// ---- POUs/P70_Interface.TcPOU
PROGRAM P70_Interface
VAR
END_VAR

(* UI Right Dashboard Variable*)
GVL_IO.aInputState[1].0 	:= GVL_IO.aDigitalInputIO[1].0; //Maintenance Key

// GVL_IO.aInputState[1].1		:= P92_Maintenance.bReactorCabinetLamp; //Reactor Cabinet Lamp
// GVL_IO.aInputState[1].2		:= P92_Maintenance.bGasCabinetLamp; // Gas Cabinet Lamp
// GVL_IO.aInputState[1].3		:= P92_Maintenance.bPowerDistributeLamp; // Power Cabinet Lamp
GVL_IO.aInputState[1].1		:= GVL_IO.aDigitalOutputIO[2].5; //Reactor Cabinet Lamp
GVL_IO.aInputState[1].2		:= GVL_IO.aDigitalOutputIO[2].6; // Gas Cabinet Lamp
GVL_IO.aInputState[1].3		:= GVL_IO.aDigitalOutputIO[2].7; // Power Cabinet Lamp

GVL_IO.aInputState[1].4 	:= GVL_IO.aDigitalInputIO[2].0; //CDA Alarm Switch
GVL_IO.aInputState[1].5		:= GVL_IO.aDigitalInputIO[2].1; //Water Flow Sensor

// GVL_IO.aInputState[1].6 	:= P11_E3508.isHeaterReady; //Induction Heater
// GVL_IO.aInputState[1].7 	:= P11_E3508.isHeaterRun; //Induction Heater
// GVL_IO.aInputState[1].8 	:= P11_E3508.isHeaterFault; //Induction Heater
GVL_IO.aInputState[1].6 	:= GVL_IO.aDigitalInputIO[2].2; //Induction Heater
GVL_IO.aInputState[1].7 	:= GVL_IO.aDigitalInputIO[2].3; //Induction Heater
GVL_IO.aInputState[1].8 	:= GVL_IO.aDigitalInputIO[2].4; //Induction Heater

// GVL_IO.aInputState[1].9	:= P15_RotationOperation.bStart_Stop; //Susceptor Rotation Motor
// GVL_IO.aInputState[1].10	:= P15_RotationOperation.bBrake_Run; //Susceptor Rotation Motor
// GVL_IO.aInputState[1].11	:= P15_RotationOperation.isRotationFault; //Susceptor Rotation Motor
GVL_IO.aInputState[1].9		:= GVL_IO.aDigitalOutputIO[3].4; //Susceptor Rotation Motor
GVL_IO.aInputState[1].10	:= GVL_IO.aDigitalOutputIO[3].5; //Susceptor Rotation Motor

// GVL_IO.aInputState[1].12 	:= P12_IQ_PLUS.isPumpWarning; //Vacuum Pump
// GVL_IO.aInputState[1].13 	:= P12_IQ_PLUS.isPumpRunning; //Vacuum Pump
// GVL_IO.aInputState[1].14 	:= P12_IQ_PLUS.isPumpFault; //Vacuum Pump
GVL_IO.aInputState[1].12 	:= GVL_IO.aDigitalInputIO[3].0; //Vacuum Pump
GVL_IO.aInputState[1].13 	:= GVL_IO.aDigitalInputIO[3].3; //Vacuum Pump
GVL_IO.aInputState[1].14 	:= GVL_IO.aDigitalInputIO[2].7; //Vacuum Pump

// GVL_IO.aInputState[1].15	:= P92_Maintenance.bReactorCabientMagnet; //Door Sensor
GVL_IO.aInputState[1].15	:= GVL_IO.aDigitalInputIO[3].6; //Door Sensor

// GVL_IO.aInputState[2].0		:= P92_Maintenance.bGasCabinetMagnet; //Door Sensor
// GVL_IO.aInputState[2].1		:= P92_Maintenance.bPowerDistributeMagnet; //Door Sensor
GVL_IO.aInputState[2].0		:= GVL_IO.aDigitalInputIO[3].7; //Door Sensor
GVL_IO.aInputState[2].1		:= GVL_IO.aDigitalInputIO[4].0; //Door Sensor

// GVL_IO.aInputState[2].2		:= P90_Interlock.bPowerResetSwitch; //Power Reset Switch
GVL_IO.aInputState[2].2		:= GVL_IO.aDigitalInputIO[1].1; //Power Reset Switch

// GVL_IO.aInputState[2].3		:= P16_CoverOperation.bUpperLimit; //Cover Upper Limit Sensor
// GVL_IO.aInputState[2].4		:= P16_CoverOperation.bLowerLimit; //Cover Upper Limit Sensor
GVL_IO.aInputState[2].3		:= GVL_IO.aDigitalInputIO[3].4; //Cover Upper Limit Sensor
GVL_IO.aInputState[2].4		:= GVL_IO.aDigitalInputIO[3].5; //Cover Upper Limit Sensor

// GVL_IO.aInputState[2].5		:= P92_Maintenance.bSMPS24V480WFault; //SMPS
// GVL_IO.aInputState[2].6		:= P92_Maintenance.bSMPS24V72WFault;
// GVL_IO.aInputState[2].7		:= P92_Maintenance.bSMPS15VPlusFault;
// GVL_IO.aInputState[2].8		:= P92_Maintenance.bSMPS15VMinusFault;
GVL_IO.aInputState[2].5		:= NOT(GVL_IO.aDigitalInputIO[4].3); //SMPS
GVL_IO.aInputState[2].6		:= NOT(GVL_IO.aDigitalInputIO[4].4); 
GVL_IO.aInputState[2].7		:= NOT(GVL_IO.aDigitalInputIO[4].5); 
GVL_IO.aInputState[2].8		:= NOT(GVL_IO.aDigitalInputIO[4].6); 

// GVL_IO.aInputState[2].9		:= P11_E3508.bInductionHeaterCB;
GVL_IO.aInputState[2].9		:= GVL_IO.aDigitalInputIO[4].7;
// GVL_IO.aInputState[2].10	:= P14_ThermalBath.bThermalBathCB;
GVL_IO.aInputState[2].10	:= GVL_IO.aDigitalInputIO[5].0;
// GVL_IO.aInputState[2].11	:= P12_IQ_PLUS.bVacuumPumpCB;
GVL_IO.aInputState[2].11	:= GVL_IO.aDigitalInputIO[5].1;
// GVL_IO.aInputState[2].12	:= P13_LineHeater.bLineHeaterCB;
GVL_IO.aInputState[2].12	:= GVL_IO.aDigitalInputIO[5].2;
// GVL_IO.aInputState[2].13	:= P15_RotationOperation.bRotationCP;
GVL_IO.aInputState[2].13	:= GVL_IO.aDigitalInputIO[5].3;
// GVL_IO.aInputState[2].14	:= P16_CoverOperation.bCoverCP;
GVL_IO.aInputState[2].14	:= GVL_IO.aDigitalInputIO[5].4;
// GVL_IO.aInputState[2].15	:= P12_IQ_PLUS.bThrottleValveCP;
GVL_IO.aInputState[2].15	:= GVL_IO.aDigitalInputIO[5].5;

GVL_IO.aInputState[3].0		:= GVL_IO.aDigitalInputIO[5].6;
GVL_IO.aInputState[3].1		:= GVL_IO.aDigitalInputIO[5].7;

GVL_IO.aInputState[3].2		:= GVL_IO.aDigitalInputIO[6].0; //Line Heater #1
GVL_IO.aInputState[3].3		:= GVL_IO.aDigitalInputIO[6].1;
GVL_IO.aInputState[3].4		:= GVL_IO.aDigitalInputIO[6].2;
GVL_IO.aInputState[3].5		:= GVL_IO.aDigitalInputIO[6].3;
GVL_IO.aInputState[3].6		:= GVL_IO.aDigitalInputIO[6].4;
GVL_IO.aInputState[3].7		:= GVL_IO.aDigitalInputIO[6].5;
GVL_IO.aInputState[3].8		:= GVL_IO.aDigitalInputIO[6].6;
GVL_IO.aInputState[3].9		:= GVL_IO.aDigitalInputIO[6].7; //Line Heater #8
GVL_IO.aInputState[3].10	:= GVL_IO.aDigitalInputIO[8].0; //Thermal Bath Temp. Deviation Alarm #1
GVL_IO.aInputState[3].11	:= GVL_IO.aDigitalInputIO[8].2;
GVL_IO.aInputState[3].12	:= GVL_IO.aDigitalInputIO[8].4;
GVL_IO.aInputState[3].13	:= GVL_IO.aDigitalInputIO[8].6;
GVL_IO.aInputState[3].14	:= GVL_IO.aDigitalInputIO[9].0;
GVL_IO.aInputState[3].15	:= GVL_IO.aDigitalInputIO[9].2; //Thermal Bath Temp. Deviation Alarm #6

GVL_IO.aInputState[4].0		:= GVL_IO.aDigitalOutputIO[1].0; // RED - Alarm
GVL_IO.aInputState[4].1		:= GVL_IO.aDigitalOutputIO[1].1; // YELLOW - Waring
GVL_IO.aInputState[4].2		:= GVL_IO.aDigitalOutputIO[1].2; // GREEN - Running
GVL_IO.aInputState[4].3		:= GVL_IO.aDigitalOutputIO[1].3; // BLUE - Maintenance
GVL_IO.aInputState[4].4		:= GVL_IO.aDigitalOutputIO[1].4; // WHITE - Idle
GVL_IO.aInputState[4].5		:= GVL_IO.aDigitalOutputIO[1].5; // BUZZER - Alarm

GVL_IO.aInputState[4].6		:= GVL_IO.aDigitalOutputIO[4].0; // DOR Vacuum State

// GVL_IO.aInputState[4].7		:= P11_E3508.nInputAlarmBytes.7; // Temp Conroller Alarm State
// GVL_IO.aInputState[4].8		:= P11_E3508.nInputManAutoBytes.7; // Temp Controller Mode State

// P90_Interlock.bInductionHeaterMC := GVL_IO.aOutputCmd[1].0;
// P90_Interlock.bThermalBathMC := GVL_IO.aOutputCmd[1].1;
// P90_Interlock.bVacuumPumpMC := GVL_IO.aOutputCmd[1].2;
// P90_Interlock.bLineHeaterMC := GVL_IO.aOutputCmd[1].3;

// P11_E3508.bOutputManAuto := GVL_IO.aOutputCmd[1].11; //Temp Controller Mode Command
// P12_IQ_PLUS.bPumpOn := GVL_IO.aOutputCmd[1].6;P12_IQ_PLUS.nTValveMode := WORD_TO_USINT(GVL_IO.aOutputCmd[2]); //Throttle Valve Mode Setting 0:Normal 1:Close 2:Open 3:Hold 4:Reset

END_PROGRAM

// ---- POUs/P91_Monitoring.TcPOU
PROGRAM P91_Monitoring
VAR
	TimeCycle			: TON;
	i 					: INT;
	idx					: INT;
	
	(*Utility Input*)
	bUtilityFault		: BYTE;	
END_VAR

(* Read from Utility Device*)
bUtilityFault		:= GVL_IO.aDigitalInputIO[7]; // 1~5 BYTE Operation, Normally Contacted

TimeCycle(IN:=TRUE, PT:=T#100MS); // 100MS Refresh Reading Time
IF TimeCycle.Q THEN
	TimeCycle(IN:=FALSE);
	
	// Reactor Ultimate Pressure Gauge
	GVL_IO.aMonitoring_PV[1] := GVL_IO.aAnalogInputIO[27] / GVL_IO.KL3464MaxValue * 10; //10Torr, 0~10V, Cal. x10
	
	// Exhaust Pressure Gauge
	GVL_IO.aMonitoring_PV[2] := GVL_IO.aAnalogInputIO[28] / GVL_IO.KL3464MaxValue * 1000; //1,000Torr, 0~10V, Cal. x1000
	GVL_IO.aAnalogOutputIO[27] := GVL_IO.aAnalogInputIO[28]; // Panel Meter Display
	
	// Double O-Ring(DOR) Gauge
	GVL_IO.aMonitoring_PV[3] := GVL_IO.aAnalogInputIO[29] / GVL_IO.KL3464MaxValueH * 100; //100kPa, 0~5V, Cal. x100
		
	//Gas Pressure 4 : N2, 5 : H2, 6 : NH3, 7 : SiH4
	FOR i:=4 TO 7 DO
		idx := i + 29;
		GVL_IO.aMonitoring_PV[i] := GVL_IO.aAnalogInputIO[idx] / GVL_IO.KL3054MaxValue * 6.89; // Cal. 6.89 bar
	END_FOR	
	
	// Cooling Water Temperature
	GVL_IO.aMonitoring_PV[8] := GVL_IO.aAnalogInputIO[37] * 0.1; // PT100, Shower Head, Cal. 0.1
	GVL_IO.aMonitoring_PV[9] := GVL_IO.aAnalogInputIO[38] * 0.1; // PT100, Shower Head, Cal. 0.1
	
END_IF

END_PROGRAM

// ---- POUs/P92_Maintenance.TcPOU
PROGRAM P92_Maintenance
VAR
	(* Input *)
	//Light
	rTrigReactorCabinetSwitch	: R_TRIG;
	rTrigReactorCabinetMagnet 	: R_TRIG;
	fTrigReactorCabinetMagnet 	: F_TRIG;
	rTrigGasCabinetSwitch		: R_TRIG;
	rTrigGasCabinetMagnet		: R_TRIG;
	fTrigGasCabinetMagnet		: F_TRIG;

	bReactorCabinetLampSwitch : BOOL;
	bGasCabinetLampSwitch	: BOOL;
	
	bReactorCabientMagnet	: BOOL;
	bGasCabinetMagnet		: BOOL;
	bPowerDistributeMagnet	: BOOL;
	
	(* Output to Device *)
	// Cabinet Lamp
	bReactorCabinetLamp		: BOOL;
	bGasCabinetLamp			: BOOL;
	bPowerDistributeLamp	: BOOL;
	
	bSMPS24V480WFault		: BOOL;
	bSMPS24V72WFault		: BOOL;
	bSMPS15VPlusFault		: BOOL;
	bSMPS15VMinusFault		: BOOL;
	// Signal Tower
	bSignalTower			: BYTE;
	TimerSignalTower		: TON;
	bBuzzer					: BOOL;
END_VAR

(* Read from Device Value *)
//Lamp
bReactorCabientMagnet 	:= GVL_IO.aDigitalInputIO[3].6;
bGasCabinetMagnet 		:= GVL_IO.aDigitalInputIO[3].7;
bPowerDistributeMagnet	:= GVL_IO.aDigitalInputIO[4].0;

//SMPS
bSMPS24V480WFault	:= NOT(GVL_IO.aDigitalInputIO[4].3);
bSMPS24V72WFault	:= NOT(GVL_IO.aDigitalInputIO[4].4);
bSMPS15VPlusFault	:= NOT(GVL_IO.aDigitalInputIO[4].5);
bSMPS15VMinusFault	:= NOT(GVL_IO.aDigitalInputIO[4].6);

// Reactor Cabinet Lamp
rTrigReactorCabinetSwitch(CLK:=GVL_IO.aDigitalInputIO[1].2);
rTrigReactorCabinetMagnet(CLK:=GVL_IO.aDigitalInputIO[3].6);
fTrigReactorCabinetMagnet(CLK:=GVL_IO.aDigitalInputIO[3].6);
IF rTrigReactorCabinetSwitch.Q OR rTrigReactorCabinetMagnet.Q OR fTrigReactorCabinetMagnet.Q THEN
	bReactorCabinetLamp := NOT(bReactorCabinetLamp);
END_IF
// Gas Delivery Cabinet Lamp
rTrigGasCabinetSwitch(CLK:= GVL_IO.aDigitalInputIO[1].3);
rTrigGasCabinetMagnet(CLK:= GVL_IO.aDigitalInputIO[3].7);
fTrigGasCabinetMagnet(CLK:= GVL_IO.aDigitalInputIO[3].7);
IF rTrigGasCabinetSwitch.Q THEN
	bGasCabinetLamp := NOT(bGasCabinetLamp);
ELSIF fTrigGasCabinetMagnet.Q THEN
	bGasCabinetLamp := TRUE;
ELSIF rTrigGasCabinetMagnet.Q THEN
	bGasCabinetLamp := FALSE;
END_IF
// Power Distribute Unit Lamp
bPowerDistributeLamp := NOT(bPowerDistributeMagnet); //Magnet Switch

(* Buzzer On/Off *)
IF bBuzzer <> GVL_IO.aInterlockEnable[1].2 THEN
	bBuzzer := GVL_IO.aInterlockEnable[1].2;
END_IF

(* Blink Signal Tower *)
CASE GVL_IO.nCaseSignalTower OF
	1: //RED 
		TimerSignalTower(IN:=TRUE, PT:=T#500MS);
		IF TimerSignalTower.Q THEN
			TimerSignalTower(IN:=FALSE);
			IF bSignalTower = 0 THEN
				bSignalTower := 2#0000_0001; // RED
			ELSE
				bSignalTower := 0;
			END_IF
		END_IF

	2: //YELLOW 
		TimerSignalTower(IN:=TRUE, PT:=T#1S);
		IF TimerSignalTower.Q THEN
			TimerSignalTower(IN:=FALSE);
			IF bSignalTower = 0 THEN
				bSignalTower := 2#0000_0010; // YELLOW
			ELSE
				bSignalTower := 0;
			END_IF
		END_IF
	3: //GREEN
		TimerSignalTower(IN:=TRUE, PT:=T#1S);
		IF TimerSignalTower.Q THEN
			TimerSignalTower(IN:=FALSE);
			IF bSignalTower = 0 THEN
				bSignalTower := 2#0000_0100; // GREEN
			ELSE
				bSignalTower := 0;
			END_IF
		END_IF
	4: //BLUE
		bSignalTower := 2#0000_1000;
	5: //WHITE
		bSignalTower := 2#0001_0000;
END_CASE

(* Write to Device Value *)
GVL_IO.aDigitalOutputIO[2].5 	:= bReactorCabinetLamp;
GVL_IO.aDigitalOutputIO[2].6 	:= bGasCabinetLamp;
GVL_IO.aDigitalOutputIO[2].7 	:= bPowerDistributeLamp;

//SignalTower
GVL_IO.aDigitalOutputIO[1].0 	:= bSignalTower.0; //0:RED-Alarm,
GVL_IO.aDigitalOutputIO[1].1 	:= bSignalTower.1; //1:YELLOW,-Warning 
GVL_IO.aDigitalOutputIO[1].2 	:= bSignalTower.2; //2:GREEN-Running
GVL_IO.aDigitalOutputIO[1].3 	:= bSignalTower.3; //3:BLUE-Idle
GVL_IO.aDigitalOutputIO[1].4 	:= bSignalTower.4; //4:WHITE-Maint
GVL_IO.aDigitalOutputIO[1].5 	:= bBuzzer; //5:BUZZER-Alarm

END_PROGRAM

// ---- POUs/FB_ControlRampGenerator.TcPOU
FUNCTION_BLOCK FB_ControlRampGenerator
VAR_INPUT
	input : RampGeneratorInput;
END_VAR
VAR
	state : E_RampGeneratorState := E_RampGeneratorState.End;
	rampGenerator : FB_CTRL_RAMP_GENERATOR;
	rampGeneratorParams	: ST_CTRL_RAMP_GENERATOR_PARAMS := (tTaskCycleTime := T#100MS, tCtrlCycleTime := T#100MS, fVeloPos := 0, fVeloNeg := 0);
END_VAR
VAR_OUTPUT
	rControlValue	: LREAL := 0;
	targetValueReached : BOOL := FALSE;
	isError : BOOL;
	eErrorID : E_CTRL_ERRORCODES;
END_VAR

IF input.restart = TRUE AND 0 <= input.rampTime AND rControlValue <> input.targetValue THEN
	state := E_RampGeneratorState.Init;
	input.restart := FALSE;
END_IF
	
CASE state OF
	E_RampGeneratorState.Init:
		IF 0 < input.rampTime THEN
			rampGeneratorParams.fVeloPos			:= ABS(input.targetValue - rControlValue) / input.rampTime * 0.1; (* in units per second *)
			rampGeneratorParams.fVeloNeg			:= rampGeneratorParams.fVeloPos; (* in units per second *)
			rampGenerator(bEnable := TRUE, fStart := rControlValue, fTarget:= input.targetValue, fOut => rControlValue, bValueReached => targetValueReached, bError => isError, eErrorID => eErrorID, stParams := rampGeneratorParams);
		ELSIF input.rampTime = 0 THEN
			rampGenerator(bEnable := FALSE, stParams := rampGeneratorParams);
			rampGeneratorParams.fVeloPos			:= input.targetValue; (* in units per second *)
			rampGeneratorParams.fVeloNeg			:= rampGeneratorParams.fVeloPos; (* in units per second *)
			rampGenerator(bEnable := TRUE, fStart := input.targetValue, fTarget:= input.targetValue, fOut => rControlValue, bValueReached => targetValueReached, bError => isError, eErrorID => eErrorID, stParams := rampGeneratorParams);
		END_IF
		state := E_RampGeneratorState.Run;
	
	E_RampGeneratorState.Run:
		rampGenerator(bEnable := TRUE, stParams := rampGeneratorParams, fOut => rControlValue, bValueReached => targetValueReached, bError => isError, eErrorID => eErrorID, stParams := rampGeneratorParams);
		IF targetValueReached = TRUE THEN
			state := E_RampGeneratorState.End;
		END_IF
		
	E_RampGeneratorState.End:
		rampGenerator(bEnable := FALSE, stParams := rampGeneratorParams, fOut => rControlValue);
END_CASE

END_FUNCTION_BLOCK

// ---- FUNTION/CheckRangeUnsigned.TcPOU
// Implicitly generated code : DO NOT EDIT
FUNCTION CheckRangeUnsigned : UDINT
VAR_INPUT
	value, lower, upper: UDINT;
END_VAR

// Implicitly generated code : Only an Implementation suggestion
{noflow}
IF (value < lower) THEN
	CheckRangeUnsigned := lower;
ELSIF(value > upper) THEN
	CheckRangeUnsigned := upper;
ELSE
	CheckRangeUnsigned := value;
END_IF
{flow}

END_FUNCTION

// ---- POUs/FB_OverLimitCheck.TcPOU
//*********************************************************************
// Function Block: FB_OverLimitCheck
// Description: 각 디바이스의 범위 초과 알람을 처리합니다.
// bEnable이 TRUE일 때만 알람 로직이 활성화됩니다.
//*********************************************************************
FUNCTION_BLOCK FB_OverLimitCheck
VAR_INPUT
	bAlarmEnable	: BOOL; //디바이스 활성화/비활성화 (TRUE = 활성화)
	bWarningEnable	: BOOL;
	fCurrentValue 	: REAL; //현재값
	fAlarmTreshold	: REAL; //알람 허용 임계값
	fWarningTreshold : REAL; //경고 허용 임계값
	tAlarmDelay		: TIME; //지연 시간
END_VAR
VAR_OUTPUT
	bAlarm			: BOOL; //허용 값 초과 경고 발생
	bWarning		: BOOL; //허용 값 초과 주의 발생
END_VAR
VAR
	//내부 변수 (인스턴스별로 독립적)
	fbAlarmTimer 		: TON;
	fbWarningTimer 	: TON;
 	bAlarmCondition 	: BOOL;
	bWarningCondition 	: BOOL; 
END_VAR

// bAlarmEnable이 TRUE일 때만 알람 로직 실행
IF bAlarmEnable THEN
	//허용값 알람 로직(지연 시간 적용)
	IF fCurrentValue > fAlarmTreshold THEN
		bAlarmCondition := TRUE;
	ELSE
		bAlarmCondition := FALSE;
	END_IF
	fbAlarmTimer(IN:=bAlarmCondition, PT:=tAlarmDelay);
	bAlarm := fbAlarmTimer.Q;
ELSE
	// bEnable이 FALSE일 경우, 모든 알람 및 타이머를 비활성화/리셋
    // Q 출력을 FALSE로 강제하고, IN 입력을 FALSE로 설정하여 타이머를 리셋합니다.
	bAlarm := FALSE;
	fbAlarmTimer(IN := FALSE, PT := tAlarmDelay); // 타이머 리셋
	bAlarmCondition := FALSE; // 조건 플래그도 리셋
END_IF

// bWarningEnable이 TRUE일 때만 알람 로직 실행
IF bWarningEnable THEN
	//허용값 주의 로직(지연 시간 적용)
	IF (fCurrentValue > fWarningTreshold) AND (fCurrentValue <= fAlarmTreshold ) THEN
		bWarningCondition := TRUE;
	ELSE
		bWarningCondition := FALSE;
	END_IF
	fbWarningTimer(IN:=bWarningCondition, PT:=tAlarmDelay);
	bWarning := fbWarningTimer.Q;
ELSE
	// bEnable이 FALSE일 경우, 모든 알람 및 타이머를 비활성화/리셋
    // Q 출력을 FALSE로 강제하고, IN 입력을 FALSE로 설정하여 타이머를 리셋합니다.
	bWarning := FALSE;
	fbWarningTimer(IN := FALSE, PT := tAlarmDelay); // 타이머 리셋
	bWarningCondition := FALSE; // 조건 플래그도 리셋
END_IF

END_FUNCTION_BLOCK
